# EPICS autosave request: CARSApp/Db/CARS_motor_positions.req
# FILE... CARS_motor_positions.req
$(P)$(M).DVAL
$(P)$(M).OFF
